// TIA Portal V18 export
TYPE "KukaRobot_HMI"
// stored: IsFailsafeCompliant false
   STRUCT
      PGNO_PBIT : USInt;   // First bit of program no.\程序编号
      EXT_START : Bool;   // Program start\程序启动
      MOVE_ENABLE : Bool;   // Motion enable\运行开通
      CONF_MESS : Bool;   // Error comfirmation\错误确认
      DRIVES_OFF : Bool;   // Drives off(inverse)\驱动装置关闭
      DRIVES_ON : Bool;   // Drives on\驱动装置接通
      I_O_ACT : Bool;   // Activate interface\激活接口
      RC_RDY1 : Bool;   // Controller ready\控制器就绪
      ALARM_STOP : Bool;   // Alarm stop active, Emergency stop circuit close\紧急关断环路关闭
      USER_SAF : Bool;   // User Safety switch closed, Operator safety closed\操作人员防护装置关闭
      PERI_RDY : Bool;   // Drives ready\驱动装置处于待机运行状态
      ROB_CAL : Bool;   // Robot calibrated\机器人已校准
      I_O_ACTCONF : Bool;   // Interface active\接口激活
      STOPMESS : Bool;   // Stop Message, Collective fault \集合故障=停止信息
      ALARM_STOP_INTERN : Bool;   // Internal emergency stop\内部紧急关断
      PGNO_FBIT_REFL : USInt;   // First bit for program mirroring\程序镜像
      PRO_ACT : Bool;   // Program active\程序激活
      APPL_RUN : Bool;   // Application running\应用程序正在运行
      PRO_MOVE : Bool;   // Program motion active\程序移动激活
      IN_HOME : Bool;   // In home position\位于起始位置
      ON_PATH : Bool;   // Robot on path\机器人在轨迹上
      NEAR_POSRET : Bool;   // Robot near path\机器人在轨迹附近
      T1 : Bool;   // Test1 mode\测试1模式
      T2 : Bool;   // Test2 mode\测试2模式
      AUT : Bool;   // Automatic mode\自动模式
      EXT : Bool;   // Automatic external mode\外部自动模式
      TaskMode : USInt;
      PartType : USInt;
      SpeedSet : USInt;
      HomeSeqStart : Bool;
      AutoCycleStart : Bool;
      CurrentMode : USInt;
      CurrentPartType : USInt;
      SpeedActual : USInt;
      ProgramSequence : USInt;
      WaitForHomeSeqStart : Bool;
      GoHomeFail : Bool;
      HomeSeqOK : Bool;
      WaitForAutoCycleStart : Bool;
      iTaskMode : USInt;
      iPartType : USInt;
      iSpeedValue : USInt;
      iPGNO : USInt;   // Robot Program number
      AutoStart : Bool;
      SrartHome : Bool;
      StartAutoCycle : Bool;
      Ready : Bool;
      StartComplete : Bool;
      StartUpTimeOut : Bool;
      Warning : Bool;
      Error : Bool;
      ErrorCode : Int;
      Seconds : Int;
      Minute : Int;
      Hours : DInt;
      CountPulse : Bool;
      StartSeq : Int;
   END_STRUCT;
END_TYPE
